// TIA Portal V18 export
ORGANIZATION_BLOCK "13-Laser Measure"   // OB132, LAD, ProgramCycle
TITLE = Laser / "Main Program Sweep (Cycle)"
{ S7_Optimized_Access := 'TRUE' }
VERSION : 0.1
// stored: AutoNumber true, IsIECCheckEnabled false, SetENOAutomatically false
   VAR_INPUT
      Initial_Call : Bool;   // Initial call of this OB
      Remanence : Bool;   // =True, if remanent data are available
   END_VAR
   VAR_TEMP
      "Laser NormScale" : Real;
   END_VAR
BEGIN

REGION Network 1: Laser
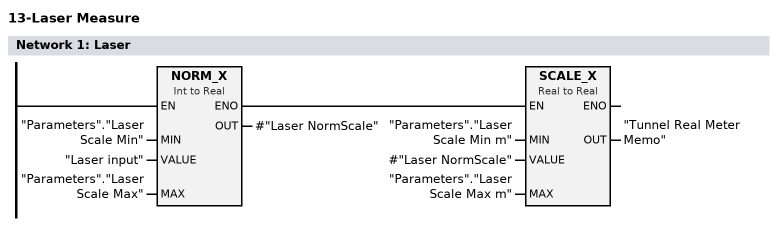
   RUNG wire#powerrail
      { S7_Templates := "[SrcType := Int, DestType := Real]" } Normalize(min := "Parameters"."Laser Scale Min", value := "Laser input", max := "Parameters"."Laser Scale Max", out => #"Laser NormScale")
      { S7_Templates := "[SrcType := Real, DestType := Real]" } Scale(min := "Parameters"."Laser Scale Min m", value := #"Laser NormScale", max := "Parameters"."Laser Scale Max m", out => "Tunnel Real Meter Memo")
   END_RUNG
   // the same network as SCL:
   #"Laser NormScale" := NORM_X(MIN := "Parameters"."Laser Scale Min", VALUE := "Laser input", MAX := "Parameters"."Laser Scale Max");
   "Tunnel Real Meter Memo" := SCALE_X(MIN := "Parameters"."Laser Scale Min m", VALUE := #"Laser NormScale", MAX := "Parameters"."Laser Scale Max m");
END_REGION
END_ORGANIZATION_BLOCK
